// TIA Portal project "Format_DateTime" (V18)

(* hardware
DEVICE "S7-1200 station_1"  S7-1200 Station
   slot 0: "Rack_0"  S7-1200 Rack  Rack  V1.0
   slot 1: "PLC_1"  CPU 1214C DC/DC/DC  6ES7 214-1AG40-0XB0  V4.5
DEVICE "HMI_1"  KTP700 Basic PN
   slot 0: "HMI_1"  KTP700 Basic PN  6AV2 123-2GB03-0AX0  17.0.0.0
   slot 1: "HMI_RT_1"  KTP700 Basic PN  6AV2 123-2GB03-0AX0  17.0.0.0
   slot 5: "HMI_1.IE_CP_1"  PROFINET Interface  17.0.0.0
      slot 1: "PROFINET Interface_1"  PROFINET Interface
         slot 1: "Port_1"  Port
*)

// ===== PLC "PLC_1"  CPU 1214C DC/DC/DC =====

VAR_GLOBAL   // PLC tag table "Default tag table"
   "System_Byte" AT %MB1 : Byte;
   "FirstScan" AT %M1.0 : Bool;
   "DiagStatusUpdate" AT %M1.1 : Bool;
   "AlwaysTRUE" AT %M1.2 : Bool;
   "AlwaysFALSE" AT %M1.3 : Bool;
   "Clock_Byte" AT %MB0 : Byte;
   "Clock_10Hz" AT %M0.0 : Bool;
   "Clock_5Hz" AT %M0.1 : Bool;
   "Clock_2.5Hz" AT %M0.2 : Bool;
   "Clock_2Hz" AT %M0.3 : Bool;
   "Clock_1.25Hz" AT %M0.4 : Bool;
   "Clock_1Hz" AT %M0.5 : Bool;
   "Clock_0.625Hz" AT %M0.6 : Bool;
   "Clock_0.5Hz" AT %M0.7 : Bool;
END_VAR

// folder: DBs

DATA_BLOCK "Var_IHM"   // DB1
{ S7_Optimized_Access := 'TRUE' }
VERSION : 0.1
   VAR
      Tela_Root : Struct
         Int_Date_Time_Local : Int;
         Date_Time_Formated : String;
         Date_Time : DTL;
      END_STRUCT;
   END_VAR
BEGIN
END_DATA_BLOCK

// folder: (top level)

ORGANIZATION_BLOCK "Main"   // OB1, LAD, ProgramCycle
TITLE = "Main Program Sweep (Cycle)"
{ S7_Optimized_Access := 'TRUE' }
VERSION : 0.1
   VAR_INPUT
      Initial_Call : Bool;   // Initial call of this OB
      Remanence : Bool;   // =True, if remanent data are available
   END_VAR
BEGIN

REGION Network 1
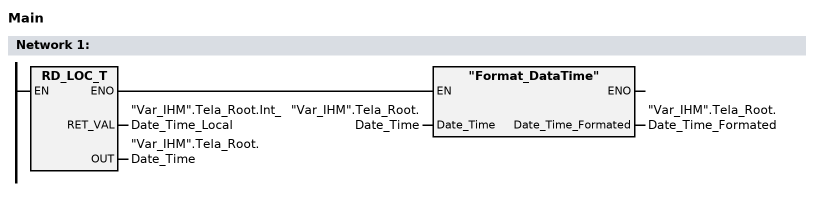
   // ENO of a box is taken as its EN; it also drops when the box reports an error
   "Var_IHM".Tela_Root.Int_Date_Time_Local := RD_LOC_T(OUT => "Var_IHM".Tela_Root.Date_Time);
   "Format_DataTime"(Date_Time := "Var_IHM".Tela_Root.Date_Time,
                     Date_Time_Formated => "Var_IHM".Tela_Root.Date_Time_Formated);
END_REGION
END_ORGANIZATION_BLOCK

// folder: FCs

FUNCTION "Format_DataTime" : Void   // FC1, SCL
TITLE = Ezequiel
{ S7_Optimized_Access := 'TRUE' }
VERSION : 0.1
// Formata data e hora para o padrao DD/MM/YYYY  HH:MM:SS
   VAR_INPUT
      Date_Time : DTL;
   END_VAR
   VAR_OUTPUT
      Date_Time_Formated : String;
   END_VAR
   VAR_TEMP
      YEAR : String;
      MONTH : String;
      DAY : String;
      HOUR : String;
      MINUTE : String;
      SECOND : String;
      "DATE" : String;
      "TIME" : String;
   END_VAR
BEGIN
   #YEAR := UINT_TO_STRING(#Date_Time.YEAR);
   #YEAR := RIGHT(IN := #YEAR, L := 4);
   #MONTH := USINT_TO_STRING(#Date_Time.MONTH);

   IF #Date_Time.MONTH >= 10 THEN
       #MONTH := RIGHT(IN := #MONTH, L := 2);
   ELSE
       #MONTH := RIGHT(IN := #MONTH, L := 1);
       #MONTH := CONCAT(IN1 := '0', IN2 := #MONTH);
   END_IF;

   #DAY := USINT_TO_STRING(#Date_Time.DAY);

   IF #Date_Time.DAY >= 10 THEN
       #DAY := RIGHT(IN := #DAY, L := 2);
   ELSE
       #DAY := RIGHT(IN := #DAY, L := 1);
       #DAY := CONCAT(IN1 := '0', IN2 :=#DAY);
   END_IF;


   #HOUR := USINT_TO_STRING(#Date_Time.HOUR);

   IF #Date_Time.HOUR >= 10 THEN
       #HOUR := RIGHT(IN := #HOUR, L := 2);
   ELSE
       #HOUR := RIGHT(IN := #HOUR, L := 1);
   END_IF;

   #MINUTE := USINT_TO_STRING(#Date_Time.MINUTE);

   IF #Date_Time.MINUTE >= 10 THEN
       #MINUTE := RIGHT(IN := #MINUTE, L := 2);
   ELSE
       #MINUTE := RIGHT(IN := #MINUTE, L := 1);
       #MINUTE := CONCAT(IN1 := '0', IN2 := #MINUTE);
   END_IF;

   #SECOND := USINT_TO_STRING(#Date_Time.SECOND);

   IF #Date_Time.SECOND >= 10 THEN
       #SECOND := RIGHT(IN := #SECOND, L := 2);
   ELSE
       #SECOND := RIGHT(IN := #SECOND, L := 1);
       #SECOND := CONCAT(IN1 := '0', IN2 := #SECOND);
   END_IF;

   #DATE := CONCAT(IN1 := #DAY, IN2 := '/');
   #DATE := CONCAT(IN1 := #DATE, IN2 := #MONTH);
   #DATE := CONCAT(IN1 := #DATE, IN2 := '/');
   #DATE := CONCAT(IN1 := #DATE, IN2 := #YEAR);
   #DATE := CONCAT(IN1 := #DATE, IN2 := ' ');
   #TIME := CONCAT(IN1 := #HOUR, IN2 := ':');
   #TIME := CONCAT(IN1 := #TIME, IN2 := #MINUTE);
   #TIME := CONCAT(IN1 := #TIME, IN2 := ':');
   #TIME := CONCAT(IN1 := #TIME, IN2 := #SECOND);

   #Date_Time_Formated := CONCAT(IN1 := #DATE, IN2 := #TIME);
END_FUNCTION

(* ===== HMI "HMI_RT_1" =====
system functions are stored by id; their names below are inferred from use
connection "HMI_Connection_1": ETHERNET, SMART_S7_1200_OMS

HMI tags "Default tag table"
   "Tag_ScreenNumber" : UInt, internal
   "Var_IHM_Tela_Root_Date_Time_Formated" : String[254] = PLC Var_IHM.Tela_Root.Date_Time_Formated, 1 s

Template "Template_1" 800x480
   Button "Alarms" at 714,429 size 71x50; TextOff 'Alarms'; PictureOff "AlarmDisplay_KTP700_Basic_PN_TR"; PictureOn "AlarmDisplay_KTP700_Basic_PN_TR"
      on Release: function_ef3f5d25("Alarm window_Unacknowledged", -1)
   Button "Template_Button" at 614,429 size 71x50; TextOff 'Text'
   Button "Template_Button_1" at 514,429 size 71x50; TextOff 'Text'
   Button "Template_Button_2" at 414,429 size 71x50; TextOff 'Text'
   Button "Template_Button_3" at 314,429 size 71x50; TextOff 'Text'
   Button "Template_Button_4" at 214,429 size 71x50; TextOff 'Text'
   Button "Template_Button_5" at 114,429 size 71x50; TextOff 'Text'
   Button "Start screen" at 14,429 size 71x50; TextOff 'Start screen'; PictureOff "NavigateHome_KTP700_Basic_PN_TR"; PictureOn "NavigateHome_KTP700_Basic_PN_TR"
      on Release: ActivateScreen("Root screen", 0)
   SymbolicIOField "Symbolic_IO_Field_Screen" at 93,9 size 600x33; TextOff '0'; TextOn '1'; TextList "TextList_ScreenNames"
      ProcessValue <- "Tag_ScreenNumber"
      on Change: ActivateScreenByNumber("Tag_ScreenNumber", 0)
   DateTimeField "HmiScreenItemData" at 695,25 size 105x25
   DateTimeField "HmiScreenItemData_1" at 695,0 size 105x25
   GraphicView "Logo" at 0,0 size 91x51; Picture "Logo of HMI_1"

screen "Root screen" 800x480, template "Template_1"
   on GenerateScreen: SetTag("Tag_ScreenNumber", 1)
   Button "HmiScreenItemData_1" at 17,49 size 159x47; TextOff 'System screens'; PictureOff "Navigates to System screens for KTP700 Basic+ PN 17.0.0.0"; PictureOn "Navigates to System screens for KTP700 Basic+ PN 17.0.0.0"
      on Release: ActivateScreen("System screens", 0)
   IOField "Template_I/O field_6" at 299,186 size 149x32; FormatPattern ????????????????????????????????????????
      ProcessValue <- "Var_IHM_Tela_Root_Date_Time_Formated"

screen "System screens" 800x480, template "Template_1"
   on GenerateScreen: SetTag("Tag_ScreenNumber", 2)
   Button "Back" at 1,52 size 159x47; TextOff 'Back'
      on Release: ActivateScreen("Root screen", 0)
   Button "HmiScreenItemData" at 36,146 size 159x47; TextOff 'SIMATIC PLC system diagnos...'; PictureOff "Navigates to SIMATIC PLC system diagnostics for KTP700 Basic+ PN 17.0.0.0"; PictureOn "Navigates to SIMATIC PLC system diagnostics for KTP700 Basic+ PN 17.0.0.0"
      on Release: ActivateScreen("SIMATIC PLC system diagnostics", 0)
   Button "HmiScreenItemData_1" at 36,205 size 159x47; TextOff 'Project information'; PictureOff "Navigates to Project information for KTP700 Basic+ PN 17.0.0.0"; PictureOn "Navigates to Project information for KTP700 Basic+ PN 17.0.0.0"
      on Release: ActivateScreen("Project information", 0)
   Button "HmiScreenItemData_2" at 36,264 size 159x47; TextOff 'User administration'; PictureOff "Navigates to User administration for KTP700 Basic+ PN 17.0.0.0"; PictureOn "Navigates to User administration for KTP700 Basic+ PN 17.0.0.0"
      on Release: ActivateScreen("User administration", 0)
   Button "HmiScreenItemData_3" at 36,323 size 159x47; TextOff 'System information'; PictureOff "Navigates to System information for KTP700 Basic+ PN 17.0.0.0"; PictureOn "Navigates to System information for KTP700 Basic+ PN 17.0.0.0"
      on Release: ActivateScreen("System information", 0)

screen "SIMATIC PLC system diagnostics" 800x480, template "Template_1"
   on GenerateScreen: SetTag("Tag_ScreenNumber", 3)
   SysDiagControl "HmiScreenItemData" at 1,100 size 796x321
   Button "Back" at 1,52 size 159x47; TextOff 'Back'
      on Release: ActivateScreen("System screens", 0)

screen "Project information" 800x480, template "Template_1"
   on GenerateScreen: SetTag("Tag_ScreenNumber", 4)
   TextField "HmiScreenItemData" at 35,102 size 171x28; Text 'Project name:'
   TextField "HmiScreenItemData_1" at 241,102 size 524x28; Text 'Format_Time'
   TextField "HmiScreenItemData_2" at 35,132 size 171x28; Text 'Created on:'
   TextField "HmiScreenItemData_3" at 241,132 size 524x28; Text '8/29/2024 8:20:00 AM'
   TextField "HmiScreenItemData_4" at 35,162 size 171x28; Text 'Author:'
   TextField "HmiScreenItemData_5" at 241,162 size 524x28; Text 'Ezequiel'
   TextField "HmiScreenItemData_6" at 35,192 size 171x28; Text 'Description:'
   TextField "HmiScreenItemData_7" at 241,192 size 524x28; Text '(not configured)'
   Button "Back" at 1,52 size 159x47; TextOff 'Back'
      on Release: ActivateScreen("System screens", 0)

screen "User administration" 800x480, template "Template_1"
   on GenerateScreen: SetTag("Tag_ScreenNumber", 5)
   UserView "HmiScreenItemData" at 1,100 size 796x321
   Button "Back" at 1,52 size 159x47; TextOff 'Back'
      on Release: ActivateScreen("System screens", 0)

screen "System information" 800x480, template "Template_1"
   on GenerateScreen: SetTag("Tag_ScreenNumber", 6)
   TextField "HmiScreenItemData" at 35,102 size 171x28; Text 'HMI device type:'
   TextField "HmiScreenItemData_1" at 241,102 size 524x28; Text 'KTP700 Basic+ PN 17.0.0.0'
   TextField "HmiScreenItemData_2" at 35,132 size 171x28; Text 'Connection:'
   TextField "HmiScreenItemData_3" at 241,132 size 524x28; Text 'PROFINET (X1)'
   TextField "HmiScreenItemData_4" at 35,162 size 171x28; Text 'PLC:'
   TextField "HmiScreenItemData_5" at 241,162 size 524x28; Text 'SIMATIC S7 1200'
   Button "Back" at 1,52 size 159x47; TextOff 'Back'
      on Release: ActivateScreen("System screens", 0)
*)